// TIA Portal V15.1 export
// export: Created 2024-06-21T08:40:51.6558059Z, ExportSetting WithDefaults, DisplayName Totally Integrated Automation Portal, DisplayVersion V15.1 Update 5, DisplayName TIA Portal Openness, DisplayVersion V15.1 Update 5, DisplayName SINAMICS Startdrive Advanced, DisplayVersion V15.1, DisplayName G130, G150, S120, S150, SINAMICS MV, S210, DisplayVersion V15.1, DisplayName G110M, G120, G120C, G120D, G120P, DisplayVersion V15.1, DisplayName STEP 7 Professional, DisplayVersion V15.1 Update 5, DisplayName STEP 7 Safety, DisplayVersion V15.1, DisplayName WinCC Professional, DisplayVersion V15.1 Update 5, DisplayName SIMATIC Visualization Architect, DisplayVersion V15.1
FUNCTION "F209000NCP01EstpInput" : Void   // FC7003, F_FBD
TITLE = Emergency Stop Inputs
{ S7_Optimized_Access := 'TRUE' }
AUTHOR : VCC
VERSION : 0.0.0.0
// =============================================================================
// This FC handels all Emergency Stop Inputs PLC 
// =============================================================================
// stored: AutoNumber false, IsIECCheckEnabled false, UDAEnableTagReadback false
BEGIN

REGION Network 1: **** 1 - Inputs **** 209000AK01 Reset command Input
   // Reset command Input
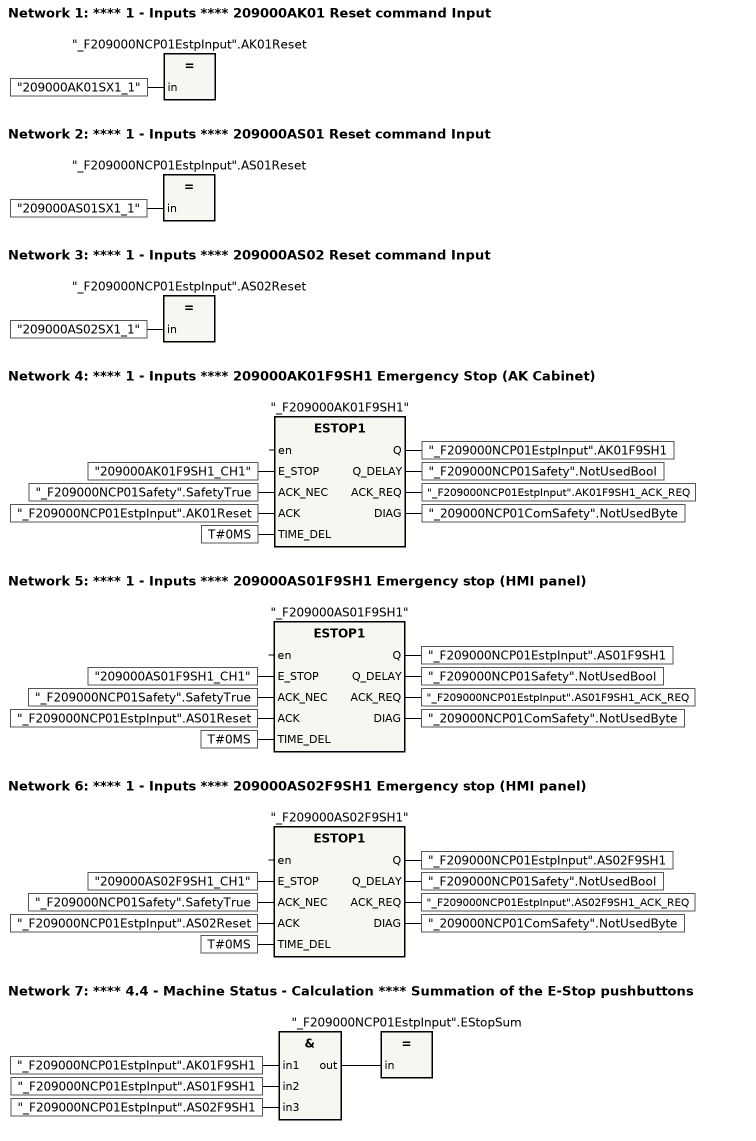
   "_F209000NCP01EstpInput".AK01Reset := "209000AK01SX1_1";
END_REGION

REGION Network 2: **** 1 - Inputs **** 209000AS01 Reset command Input
   // Reset command Input
   "_F209000NCP01EstpInput".AS01Reset := "209000AS01SX1_1";
END_REGION

REGION Network 3: **** 1 - Inputs **** 209000AS02 Reset command Input
   // Reset command Input
   "_F209000NCP01EstpInput".AS02Reset := "209000AS02SX1_1";
END_REGION

REGION Network 4: **** 1 - Inputs **** 209000AK01F9SH1 Emergency Stop (AK Cabinet)
   // Emergency Stop
   "_F209000AK01F9SH1"(E_STOP := "209000AK01F9SH1_CH1",   // ESTOP1
                       ACK_NEC := "_F209000NCP01Safety".SafetyTrue,
                       ACK := "_F209000NCP01EstpInput".AK01Reset,
                       TIME_DEL := T#0MS,
                       Q => "_F209000NCP01EstpInput".AK01F9SH1,
                       Q_DELAY => "_F209000NCP01Safety".NotUsedBool,
                       ACK_REQ => "_F209000NCP01EstpInput".AK01F9SH1_ACK_REQ,
                       DIAG => "_209000NCP01ComSafety".NotUsedByte);
END_REGION

REGION Network 5: **** 1 - Inputs **** 209000AS01F9SH1 Emergency stop (HMI panel)
   // Emergency Stop
   "_F209000AS01F9SH1"(E_STOP := "209000AS01F9SH1_CH1",   // ESTOP1
                       ACK_NEC := "_F209000NCP01Safety".SafetyTrue,
                       ACK := "_F209000NCP01EstpInput".AS01Reset,
                       TIME_DEL := T#0MS,
                       Q => "_F209000NCP01EstpInput".AS01F9SH1,
                       Q_DELAY => "_F209000NCP01Safety".NotUsedBool,
                       ACK_REQ => "_F209000NCP01EstpInput".AS01F9SH1_ACK_REQ,
                       DIAG => "_209000NCP01ComSafety".NotUsedByte);
END_REGION

REGION Network 6: **** 1 - Inputs **** 209000AS02F9SH1 Emergency stop (HMI panel)
   // Emergency Stop
   "_F209000AS02F9SH1"(E_STOP := "209000AS02F9SH1_CH1",   // ESTOP1
                       ACK_NEC := "_F209000NCP01Safety".SafetyTrue,
                       ACK := "_F209000NCP01EstpInput".AS02Reset,
                       TIME_DEL := T#0MS,
                       Q => "_F209000NCP01EstpInput".AS02F9SH1,
                       Q_DELAY => "_F209000NCP01Safety".NotUsedBool,
                       ACK_REQ => "_F209000NCP01EstpInput".AS02F9SH1_ACK_REQ,
                       DIAG => "_209000NCP01ComSafety".NotUsedByte);
END_REGION

REGION Network 7: **** 4.4 - Machine Status - Calculation **** Summation of the E-Stop pushbuttons
   // Summation of the E-Stop pushbuttons
   "_F209000NCP01EstpInput".EStopSum := "_F209000NCP01EstpInput".AK01F9SH1 AND "_F209000NCP01EstpInput".AS01F9SH1 AND "_F209000NCP01EstpInput".AS02F9SH1;
END_REGION
END_FUNCTION
